DATA_BLOCK "DB3_Super_2"
{ S7_Optimized_Access := 'FALSE' }
VERSION : 0.1
NON_RETAIN
   STRUCT
      some_1 : Bool;
      some_2 : Bool;
      som6 : Bool;
      som5 : Bool;
      som4 : Bool;
      som3 : Bool;
      som2 : Bool;
      some_3 : Bool;
      some_Int_1 : Int;
      some_bit_0 : Bool;
      some_byte_1 : Byte;
      some_bit : Bool;
      some_real : Real;
      some_bit_1 : Bool;   // some 1
      some_real_2 : Real;
      some_bit_3 : Bool;
      some_int : Int;
      wasyl : Struct   // some 2
         some_1 : Bool;
         int_1 : Int;
         bool_End : Bool;
         some : Bool;
         some2 : Bool;
         some3 : Bool;
         some4 : Bool;
         some5 : Bool;
         some6 : Bool;
         some7 : Bool;
         some8 : Bool;
         some9 : Bool;
      END_STRUCT;
      some_4 : Bool;   // some 3
      Other_Real : Real;
      some_arr : Byte;
      some_bool_2 : Bool;
      some_other_arr : Int;   // tekst some
      some_9_bool : Bool;
      other_Struct : Struct
         one : Bool;
         two : Bool;
         three : Bool;
      END_STRUCT;
      some_other : Bool;
      r1 : Bool;
      some_bool_4 : Bool;
      some_robert : Bool;
      other : Bool;
      some_Struct : Struct   // jal
         rob : Bool;
         dipper_Struct : Struct
            littleOne : Bool;
            litttleTwo : Int;
         END_STRUCT;
      END_STRUCT;
      addidas : Bool;
      kot_1 : Struct
         item_1 : Bool;
         item_2 : Bool;
      END_STRUCT;
      byte_1 : Byte;
      some_bit_2 : Bool;
      some_byte : Byte;
      some_other_bit : Bool;
      char_1 : Char;
      bool_one : Bool;
      int_44 : Int;
      sbool : Bool;
      sReal : Real;
      ssbool : Bool;
      ssInt : Int;
      sssbool : Bool;
      sssByte : Byte;
      sssReal : Real;
      arr_big : Byte;
      new_bool : Bool;
      lastStruct : Struct
         bool1 : Int;
         bool2 : Bool;
         bool3 : Bool;
         bool4 : Bool;
         d1 : Bool;
         d2 : Bool;
         d3 : Bool;
         d4 : Bool;
         d5 : Bool;
      END_STRUCT;
      newInt : Int;
   END_STRUCT;


BEGIN
   wasyl.int_1 := 0;
   wasyl.bool_End := false;
   char_1 := ' ';

END_DATA_BLOCK

